(*udt (user defined type) of Beckhoff EL2904 - 4 Point PNP Safety Type Output Terminal:
	auth. Brent Lekx-Toniolo of Toniolo Research & Development Inc.; 
	July 2010; version 1.0*)


TYPE udt_EL2904RO :
STRUCT
	Q0: BOOL;
	Q1: BOOL;
	Q2: BOOL;
	Q3: BOOL;
	InfoData: udt_ECATSlave_Status;
END_STRUCT
END_TYPE

(* stored: Version 1.1.0.1, ProductVersion 3.1.4024.9
   DUT udt_EL2904RO: Id {50c50270-4bfe-4e17-8fe3-2f2ff7ccacb2} *)
